// TIA Portal V19 export
VAR_GLOBAL   // PLC tag table "TextListId_1"
END_VAR
VAR_GLOBAL CONSTANT   // user constants
   "TEXT_LIST_ID_PN_DEV_DIAG(1)" : Int := 591;   // ID of PLC Alarm text list / SICAR: ID von SPS Alarm Textlist
   TEXT_LIST_ID_CHECKSUM : Int := 584;   // ID of PLC Alarm text list / SICAR: ID von SPS Alarm Textlist
   TEXT_LIST_ID_SMC_PD : Int := 585;   // ID of PLC Alarm text list / SICAR: ID von SPS Alarm Textlist
END_VAR
